(* LS Electric XG5000 project: Coffee_make *)
(* PLC LSPLC *)

(* Comments on direct variables
%MX1	원두리필시작
%MX2	원두부족알림
%MX3	물리필시작
%MX4	물부족알림
%MX5	우유리필시작
%MX6	우유부족알림
*)

PROGRAM NewProgram (* task: 스캔 프로그램 *)
VAR
    on AT %IX0.0.0 : BOOL;
    timer : TON;
    timer2 : TON;
    timer3 : TON;
    timer4 : TON;
    timer5 : TON;
    timer6 : TON;
    다음으로 : BOOL;
    다음으로자가유지 : BOOL;
    물 AT %MW22 : INT;
    물끓이기 : TON;
    물무게 AT %MW11 : INT;
    물무게UDINT : UDINT;
    물무게곱하기 : INT;
    물투입 : TON;
    물투입시간 : TIME;
    물투입통과 : BOOL;
    섞기 : TON;
    섞기통과 : BOOL;
    시럽무게곱하기 : INT;
    시럽우유무게UDINT : UDINT;
    시럽우유투입 : TON;
    시럽우유투입시간 : TIME;
    얼음선투입 AT %MX16 : BOOL;
    얼음선투입타이머 : TON;
    얼음선투입통과 : BOOL;
    얼음후투입 AT %MX17 : BOOL;
    얼음후투입타이머 : TON;
    얼음후투입통과 : BOOL;
    에이드액무게 : INT := 0;
    에이드투입 : BOOL := 0;
    우유 AT %MW24 : INT;
    우유뎁히기 : TON;
    우유무게 AT %MW12 : INT := 0;
    우유무게UDINT : UDINT;
    우유무게곱하기 : INT;
    우유투입 : TON;
    우유투입시간 : TIME;
    우유투입여부 : BOOL;
    우유투입통과 : BOOL;
    원두 AT %MW20 : INT;
    원두갈기 : TON;
    원두넣기 : TON;
    원두넣기시간 : TIME := T#5s;
    원두추출 : TON;
    음료제조시작 AT %IX0.0.1 : BOOL;
    음료제조완료 AT %QX0.1.0 : BOOL;
    음료제조자가유지 : BOOL;
    일단멈춰 : BOOL := 0;
    일단멈춰2 : BOOL;
    일단멈춰3 : BOOL;
    일단멈춰4 : BOOL;
    일단멈춰5 : BOOL;
    일단멈춰6 : BOOL;
    일단멈춰7 : BOOL;
    일단멈춰8 : BOOL;
    재고물 AT %MW23 : INT;
    재고우유 AT %MW25 : INT;
    재고원두 AT %MW21 : INT;
    초코시럽무게 AT %MW13 : INT;
    초코시럽무게UDINT : UDINT;
    초코시럽무게곱하기 : INT;
    초코시럽투입 : TON;
    초코시럽투입시간 : TIME;
    초코시럽투입여부 : BOOL;
    초코시럽투입통과 : BOOL;
    카페시럽무게 AT %MW14 : INT := 0;
    카페시럽무게UDINT : UDINT;
    카페시럽무게곱하기 : INT;
    카페시럽투입 : TON;
    카페시럽투입1 : TON;
    카페시럽투입2 : TON;
    카페시럽투입시간 : TIME;
    카페시럽투입여부 : BOOL;
    카페시럽투입통과 : BOOL;
    커피가레일로 : TON;
    커피끓이기시간 : TIME;
    커피무게 AT %MW10 : INT;
    커피무게UDINT : UDINT;
    커피무게곱하기 : INT;
    커피온도 AT %MW15 : INT;
    커피온도UDINT : UDINT;
    커피온도곱하기 : INT;
    커피추출 : TON;
    커피투입 : TON;
    커피투입시간 : TIME;
    커피투입시작 : BOOL;
    커피투입통과 : BOOL;
    컵구멍인지 : TON;
    컵투입 : TON;
    컵투입통과 : BOOL;
    호퍼닫기 : BOOL;
END_VAR
VAR
    _t1 : BOOL;
    _t2 : BOOL;
    _p3 : BOOL;
    _t4 : BOOL;
    _t5 : BOOL;
    _t6 : BOOL;
    _t7 : BOOL;
    _t8 : BOOL;
    _t9 : BOOL;
    _t10 : BOOL;
END_VAR

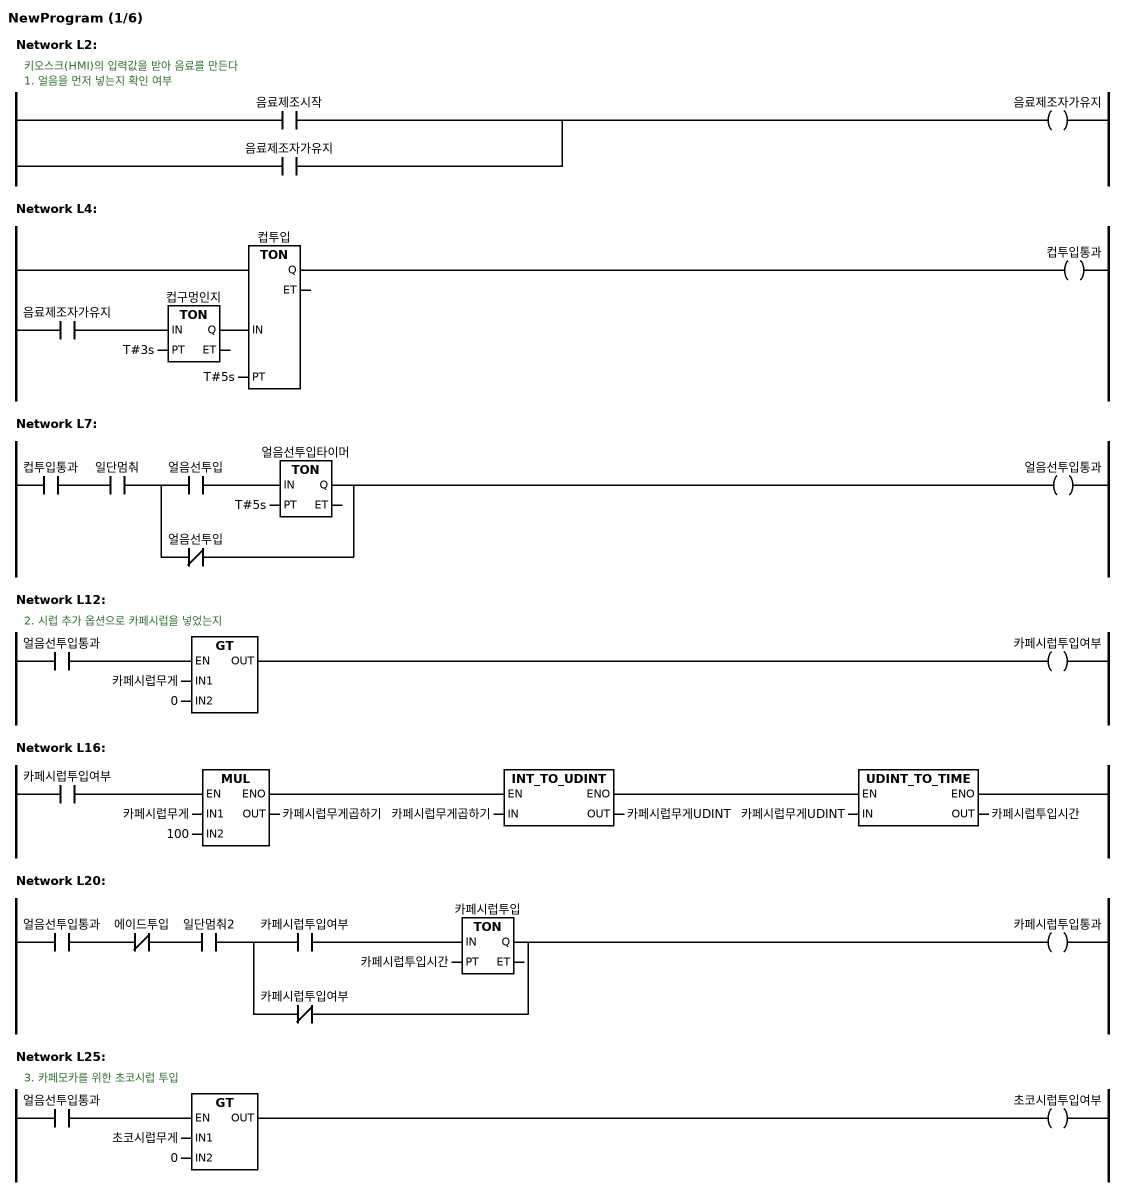
(* 키오스크(HMI)의 입력값을 받아 음료를 만든다 *)
(* 1. 얼음을 먼저 넣는지 확인 여부 *)
(* Rung L2 *)
음료제조자가유지 := 음료제조시작 OR 음료제조자가유지;
(* Rung L4 *)
컵구멍인지(IN := 음료제조자가유지, PT := T#3s);
컵투입(IN := 컵구멍인지.Q, PT := T#5s);
컵투입통과 := 컵투입.Q;
(* Rung L7 *)
얼음선투입타이머(IN := 컵투입통과 AND 일단멈춰 AND 얼음선투입, PT := T#5s);
얼음선투입통과 := 얼음선투입타이머.Q OR (컵투입통과 AND 일단멈춰 AND NOT 얼음선투입);
(* 2. 시럽 추가 옵션으로 카페시럽을 넣었는지 *)
(* Rung L12 *)
IF 얼음선투입통과 THEN _t1 := 카페시럽무게 > 0; END_IF;
카페시럽투입여부 := _t1;
(* Rung L16 *)
IF 카페시럽투입여부 THEN
    카페시럽무게곱하기 := 카페시럽무게 * 100;
    카페시럽무게UDINT := INT_TO_UDINT(카페시럽무게곱하기);
    카페시럽투입시간 := UDINT_TO_TIME(카페시럽무게UDINT);
END_IF;
(* Rung L20 *)
카페시럽투입(IN := 얼음선투입통과 AND NOT 에이드투입 AND 일단멈춰2 AND 카페시럽투입여부, PT := 카페시럽투입시간);
카페시럽투입통과 := 카페시럽투입.Q OR (얼음선투입통과 AND NOT 에이드투입 AND 일단멈춰2 AND NOT 카페시럽투입여부);
(* 3. 카페모카를 위한 초코시럽 투입 *)
(* Rung L25 *)
IF 얼음선투입통과 THEN _t2 := 초코시럽무게 > 0; END_IF;
초코시럽투입여부 := _t2;

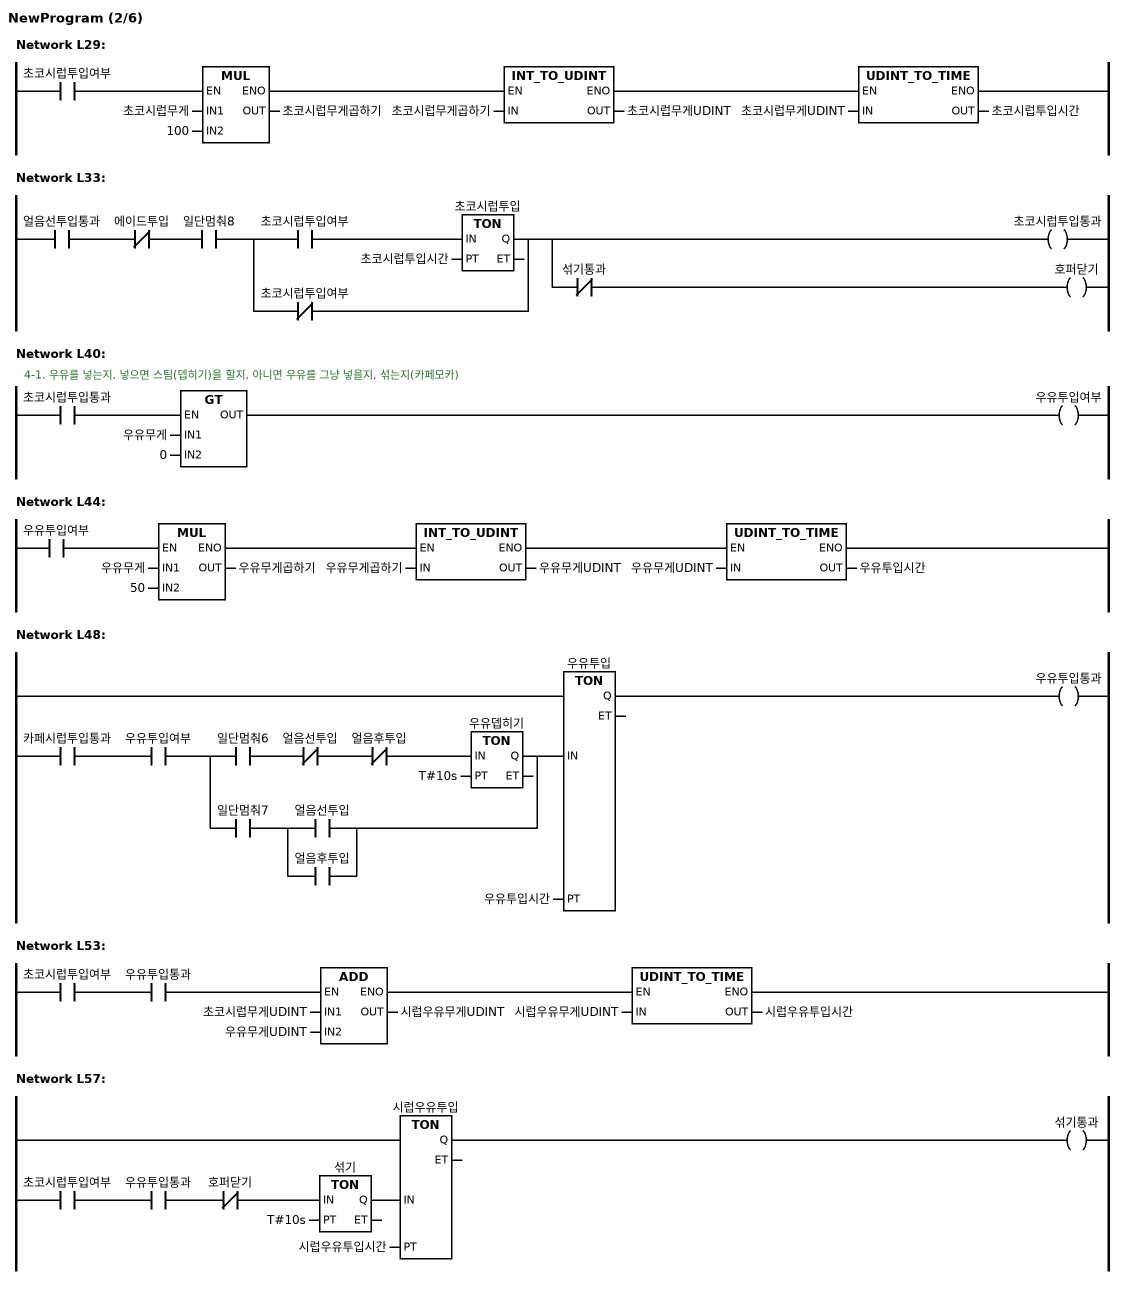
(* Rung L29 *)
IF 초코시럽투입여부 THEN
    초코시럽무게곱하기 := 초코시럽무게 * 100;
    초코시럽무게UDINT := INT_TO_UDINT(초코시럽무게곱하기);
    초코시럽투입시간 := UDINT_TO_TIME(초코시럽무게UDINT);
END_IF;
(* Rung L33 *)
초코시럽투입(IN := 얼음선투입통과 AND NOT 에이드투입 AND 일단멈춰8 AND 초코시럽투입여부, PT := 초코시럽투입시간);
_p3 := 초코시럽투입.Q OR (얼음선투입통과 AND NOT 에이드투입 AND 일단멈춰8 AND NOT 초코시럽투입여부);
초코시럽투입통과 := _p3;
호퍼닫기 := _p3 AND NOT 섞기통과;
(* 4-1. 우유를 넣는지, 넣으면 스팀(뎁히기)을 할지, 아니면 우유를 그냥 넣을지, 섞는지(카페모카) *)
(* Rung L40 *)
IF 초코시럽투입통과 THEN _t4 := 우유무게 > 0; END_IF;
우유투입여부 := _t4;
(* Rung L44 *)
IF 우유투입여부 THEN
    우유무게곱하기 := 우유무게 * 50;
    우유무게UDINT := INT_TO_UDINT(우유무게곱하기);
    우유투입시간 := UDINT_TO_TIME(우유무게UDINT);
END_IF;
(* Rung L48 *)
우유뎁히기(IN := 카페시럽투입통과 AND 우유투입여부 AND 일단멈춰6 AND NOT 얼음선투입 AND NOT 얼음후투입, PT := T#10s);
우유투입(IN := 우유뎁히기.Q OR (카페시럽투입통과 AND 우유투입여부 AND 일단멈춰7 AND (얼음선투입 OR 얼음후투입)), PT := 우유투입시간);
우유투입통과 := 우유투입.Q;
(* Rung L53 *)
IF 초코시럽투입여부 AND 우유투입통과 THEN
    시럽우유무게UDINT := 초코시럽무게UDINT + 우유무게UDINT;
    시럽우유투입시간 := UDINT_TO_TIME(시럽우유무게UDINT);
END_IF;
(* Rung L57 *)
섞기(IN := 초코시럽투입여부 AND 우유투입통과 AND NOT 호퍼닫기, PT := T#10s);
시럽우유투입(IN := 섞기.Q, PT := 시럽우유투입시간);
섞기통과 := 시럽우유투입.Q;

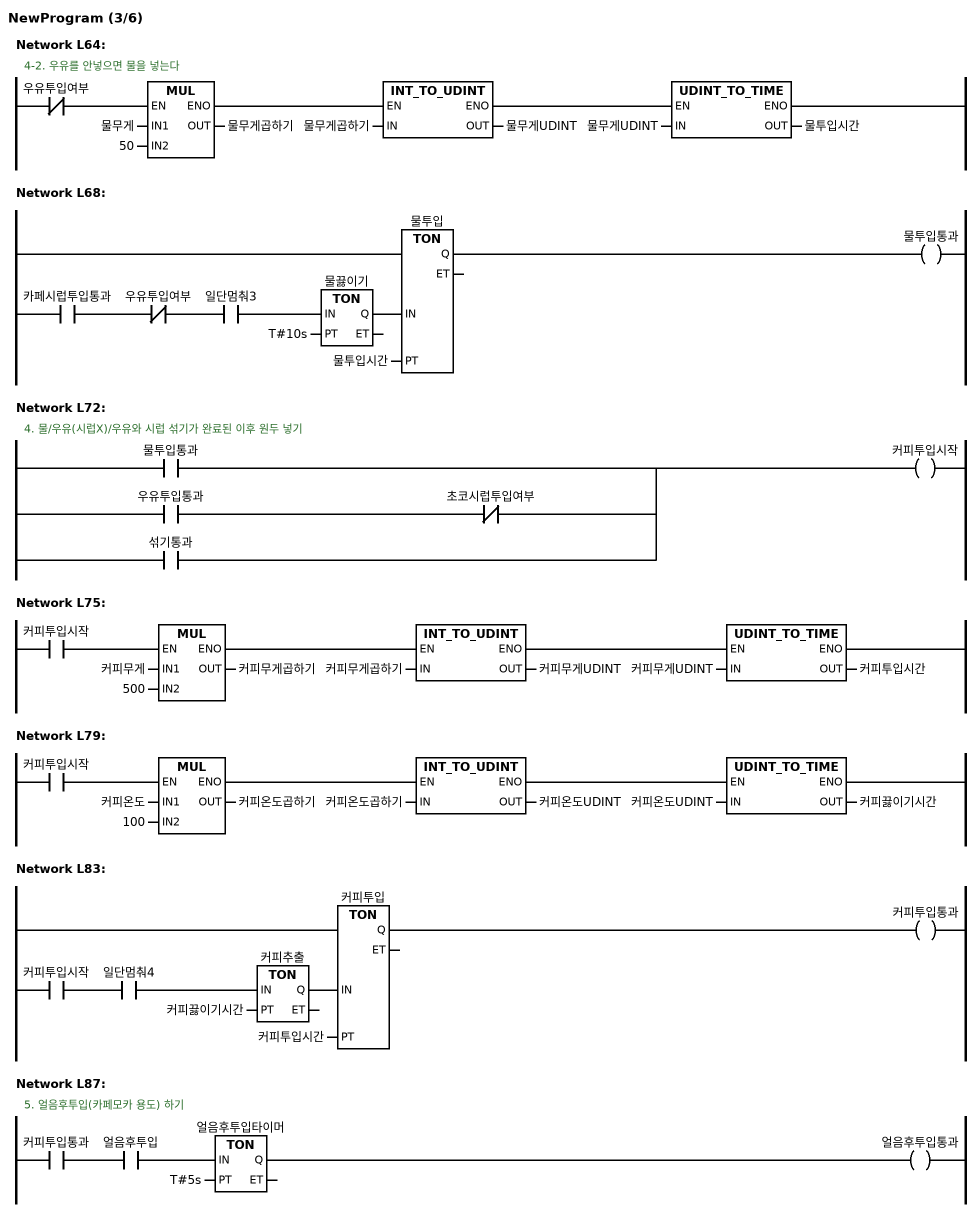
(* 4-2. 우유를 안넣으면 물을 넣는다 *)
(* Rung L64 *)
IF NOT 우유투입여부 THEN
    물무게곱하기 := 물무게 * 50;
    물무게UDINT := INT_TO_UDINT(물무게곱하기);
    물투입시간 := UDINT_TO_TIME(물무게UDINT);
END_IF;
(* Rung L68 *)
물끓이기(IN := 카페시럽투입통과 AND NOT 우유투입여부 AND 일단멈춰3, PT := T#10s);
물투입(IN := 물끓이기.Q, PT := 물투입시간);
물투입통과 := 물투입.Q;
(* 4. 물/우유(시럽X)/우유와 시럽 섞기가 완료된 이후 원두 넣기 *)
(* Rung L72 *)
커피투입시작 := 물투입통과 OR (우유투입통과 AND NOT 초코시럽투입여부) OR 섞기통과;
(* Rung L75 *)
IF 커피투입시작 THEN
    커피무게곱하기 := 커피무게 * 500;
    커피무게UDINT := INT_TO_UDINT(커피무게곱하기);
    커피투입시간 := UDINT_TO_TIME(커피무게UDINT);
END_IF;
(* Rung L79 *)
IF 커피투입시작 THEN
    커피온도곱하기 := 커피온도 * 100;
    커피온도UDINT := INT_TO_UDINT(커피온도곱하기);
    커피끓이기시간 := UDINT_TO_TIME(커피온도UDINT);
END_IF;
(* Rung L83 *)
커피추출(IN := 커피투입시작 AND 일단멈춰4, PT := 커피끓이기시간);
커피투입(IN := 커피추출.Q, PT := 커피투입시간);
커피투입통과 := 커피투입.Q;
(* 5. 얼음후투입(카페모카 용도) 하기 *)
(* Rung L87 *)
얼음후투입타이머(IN := 커피투입통과 AND 얼음후투입, PT := T#5s);
얼음후투입통과 := 얼음후투입타이머.Q;

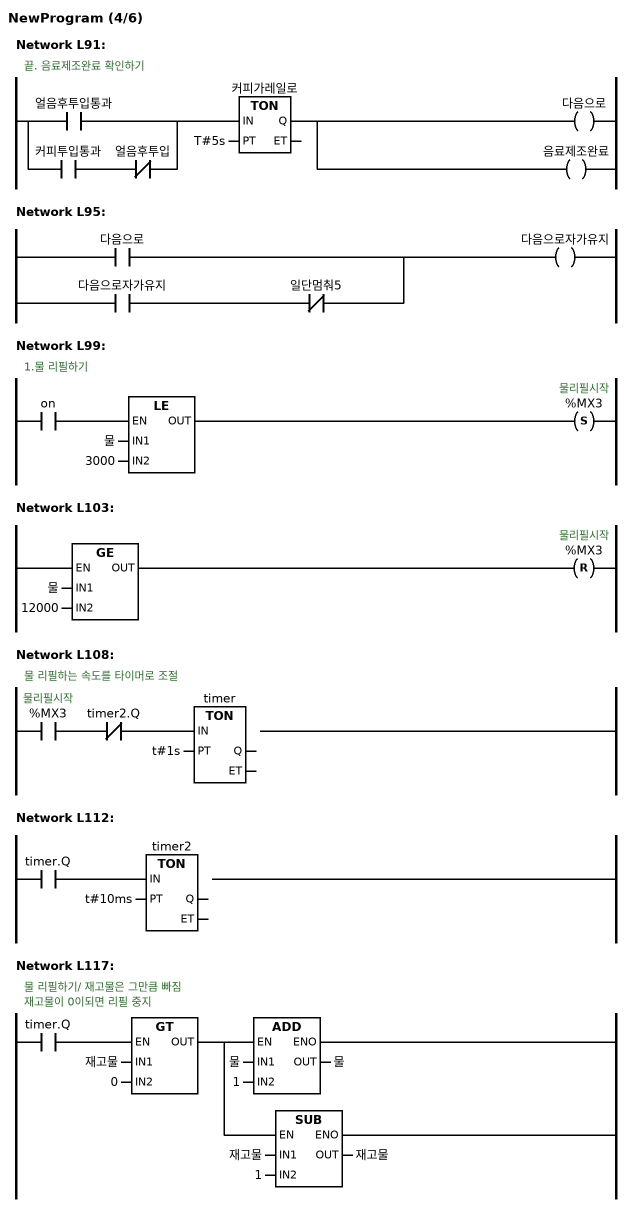
(* 끝. 음료제조완료 확인하기 *)
(* Rung L91 *)
커피가레일로(IN := 얼음후투입통과 OR (커피투입통과 AND NOT 얼음후투입), PT := T#5s);
다음으로 := 커피가레일로.Q;
음료제조완료 := 커피가레일로.Q;
(* Rung L95 *)
다음으로자가유지 := 다음으로 OR (다음으로자가유지 AND NOT 일단멈춰5);
(* 1.물 리필하기 *)
(* Rung L99 *)
IF on THEN _t5 := 물 <= 3000; END_IF;
IF _t5 THEN %MX3 := TRUE; END_IF;
(* Rung L103 *)
IF 물 >= 12000 THEN %MX3 := FALSE; END_IF;
(* 물 리필하는 속도를 타이머로 조절 *)
(* Rung L108 *)
timer(IN := %MX3 AND NOT timer2.Q, PT := t#1s);
(* Rung L112 *)
timer2(IN := timer.Q, PT := t#10ms);
(* 물 리필하기/ 재고물은 그만큼 빠짐 *)
(* 재고물이 0이되면 리필 중지 *)
(* Rung L117 *)
IF timer.Q THEN _t6 := 재고물 > 0; END_IF;
IF _t6 THEN
    물 := 물 + 1;
    재고물 := 재고물 - 1;
END_IF;

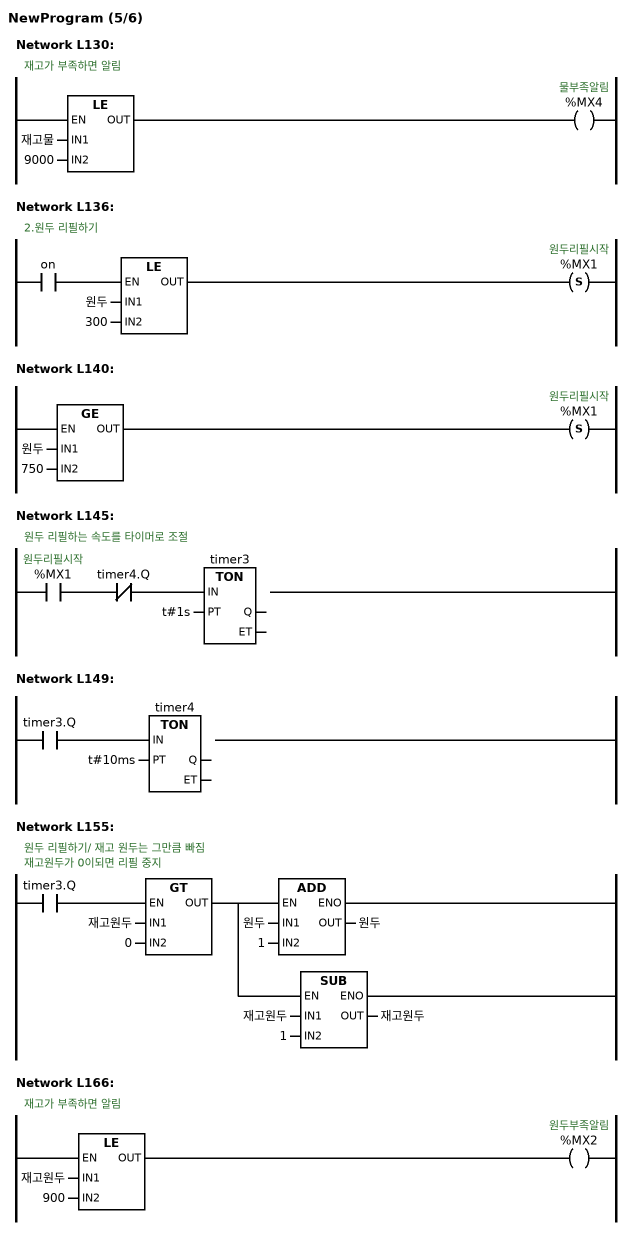
(* 재고가 부족하면 알림 *)
(* Rung L130 *)
%MX4 := 재고물 <= 9000;
(* 2.원두 리필하기 *)
(* Rung L136 *)
IF on THEN _t7 := 원두 <= 300; END_IF;
IF _t7 THEN %MX1 := TRUE; END_IF;
(* Rung L140 *)
IF 원두 >= 750 THEN %MX1 := TRUE; END_IF;
(* 원두 리필하는 속도를 타이머로 조절 *)
(* Rung L145 *)
timer3(IN := %MX1 AND NOT timer4.Q, PT := t#1s);
(* Rung L149 *)
timer4(IN := timer3.Q, PT := t#10ms);
(* 원두 리필하기/ 재고 원두는 그만큼 빠짐 *)
(* 재고원두가 0이되면 리필 중지 *)
(* Rung L155 *)
IF timer3.Q THEN _t8 := 재고원두 > 0; END_IF;
IF _t8 THEN
    원두 := 원두 + 1;
    재고원두 := 재고원두 - 1;
END_IF;
(* 재고가 부족하면 알림 *)
(* Rung L166 *)
%MX2 := 재고원두 <= 900;

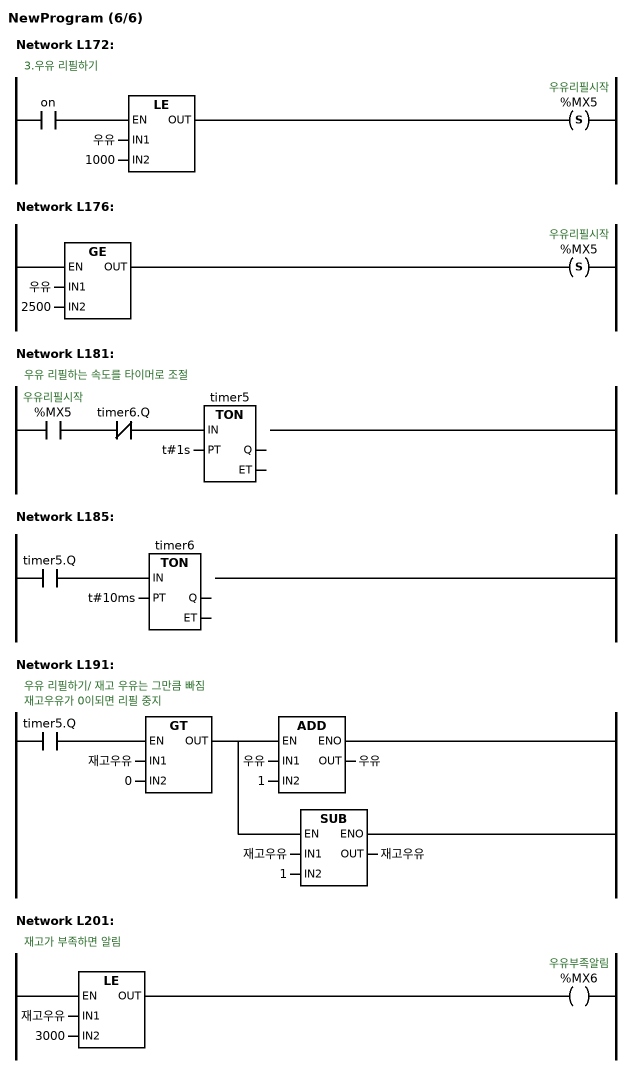
(* 3.우유 리필하기 *)
(* Rung L172 *)
IF on THEN _t9 := 우유 <= 1000; END_IF;
IF _t9 THEN %MX5 := TRUE; END_IF;
(* Rung L176 *)
IF 우유 >= 2500 THEN %MX5 := TRUE; END_IF;
(* 우유 리필하는 속도를 타이머로 조절 *)
(* Rung L181 *)
timer5(IN := %MX5 AND NOT timer6.Q, PT := t#1s);
(* Rung L185 *)
timer6(IN := timer5.Q, PT := t#10ms);
(* 우유 리필하기/ 재고 우유는 그만큼 빠짐 *)
(* 재고우유가 0이되면 리필 중지 *)
(* Rung L191 *)
IF timer5.Q THEN _t10 := 재고우유 > 0; END_IF;
IF _t10 THEN
    우유 := 우유 + 1;
    재고우유 := 재고우유 - 1;
END_IF;
(* 재고가 부족하면 알림 *)
(* Rung L201 *)
%MX6 := 재고우유 <= 3000;
END_PROGRAM